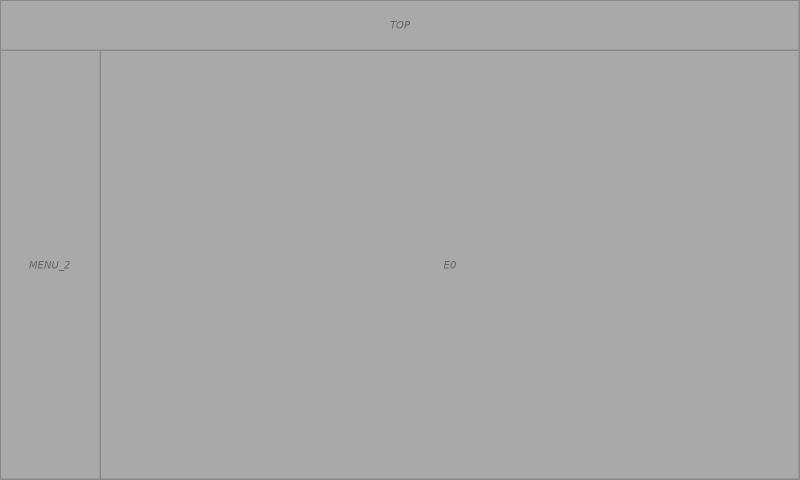
VISUALIZATION MAIN  // 800x480
    Frame (100,50 700x430)
        shows E0()
        shows E1()
        shows E2()
    Frame (0,50 100x430)
        shows MENU_2()
    Frame (0,0 800x50)
        shows TOP()
        shows MENU_2()
END_VISUALIZATION

(* stored: Version 1.1.0.1, ProductVersion 3.1.4024.15
   Visu MAIN: Id {e21716a2-9af9-455d-aa29-bbbe5337db44} *)
